FUNCTION_BLOCK PositionTrigger EXTENDS Objective

VAR
    internalPosition    	 : LREAL;
    internalTriggerDirection 	 : Tc2_MC2.MC_Direction;
    internalMoverPassedPosition : BOOL;
    internalCurrentMover     	 : POINTER TO Mover;
	internalLastMoverPassedPosition		: BOOL;
	internalTrack				: REFERENCE TO TRACK;
    moverLastPos              	: ARRAY[1..GVL.NUM_MOVERS] OF LREAL; // Positions of tracked movers from last cycle
	moverInitialized			: ARRAY [1..GVL.NUM_MOVERS] OF BOOL; // first scan-like flag to prevent erronious triggers on first scan
	
	lastCallMuteCurrent: LREAL;
	internalInterarrivalTimer			: TON;
	internalStatisticsReset				: BOOL;
END_VAR
VAR_OUTPUT
	Statistics							: PositionTriggerStats_typ;
END_VAR

{attribute 'monitoring' := 'call'}
PROPERTY CurrentMover : REFERENCE TO Mover
GET


CurrentMover						REF= internalCurrentMover^;
CurrentMover.SourceInstancePath		:= THIS^.InstancePath;

// If the Trigger has no CurrentMover, then return an imposter ErrorMover,
// whose method calls all trigger an error message
IF __ISVALIDREF(CurrentMover) = FALSE THEN
    ErrorMover.SourceInstancePath := THIS^.InstancePath;
    CurrentMover                  REF= ErrorMover;
END_IF
END_GET
END_PROPERTY

METHOD Cyclic : BOOL
VAR_INPUT
END_VAR
VAR
	
    i                       	: UDINT;	
	currentIsRegistered			: BOOL;
	moverTrackId				: INT;
	positionDifference			: LREAL;
	modTrackPosition			: LREAL;
	rolloverOccured				: BOOL;
	
END_VAR
VAR_INST

	velocityCount				: UDINT;
	velocitySum					: LREAL;
	internalRingBufferIDX		: UDINT;
	alphaEMA					: LREAL;

END_VAR
currentIsRegistered		:= FALSE;

FOR i := 1 TO GVL.NUM_MOVERS DO
    IF internalTrackedMovers[i] <> 0 AND_THEN internalTrackedMovers[i]^.IsTrackReady AND internalTrackedMovers[i]^.CurrentTrack <> 0 THEN
		moverTrackId := internalTrackedMovers[i]^.CurrentTrack^.Id;
		IF (moverTrackId = internalTrack.Id) THEN
			
			// last position is invalid on first scan, set it to the current position to avoid a false trigger on the first scan
			IF NOT moverInitialized[i] THEN
				moverInitialized[i] := TRUE;
				moverLastPos[i] := modTrackPosition;
			END_IF
		
			// Determine if a position rollover occured in the last cycle
			modTrackPosition := MODABS( internalTrackedMovers[i]^.TrackInfo.TrackPosition, internalTrackedMovers[i]^.CurrentTrack^.Length);
			positionDifference := moverLastPos[i] - modTrackPosition;			
			rolloverOccured := ABS( positionDifference ) > ( internalTrackedMovers[i]^.CurrentTrack^.Length / 2 );
			
			// and if so, modify the stored last position values to be nonmodulo to compensate
			IF rolloverOccured AND positionDifference > 0 THEN
				moverLastPos[i]		:= moverLastPos[i] - internalTrackedMovers[i]^.CurrentTrack^.Length;
			ELSIF rolloverOccured AND positionDifference < 0 THEN
				moverLastPos[i]		:= moverLastPos[i] + internalTrackedMovers[i]^.CurrentTrack^.Length;
			END_IF
		
			// Look for movers passing over the threshold this cycle and assign it to the
			// InternalCurrentMover output, which should latch until it is cleared
			IF TriggerDirection = MC_Positive_Direction AND moverLastPos[i] < internalPosition AND
				modTrackPosition >= internalPosition THEN
				
				// Position trigger event detected in the positive direction
				internalMoverPassedPosition		:= TRUE;
				internalCurrentMover			:= internalTrackedMovers[i];
				
			ELSIF TriggerDirection = MC_Negative_Direction AND moverLastPos[i] > internalPosition AND
				modTrackPosition <= internalPosition THEN
				
				// Position trigger event detecte in the negative direction
				internalMoverPassedPosition		:= TRUE;
				internalCurrentMover			:= internalTrackedMovers[i];
				
			END_IF
			
			
			
			// Ensure that the CurrentMover is still registered with the PositionTrigger
			IF internalCurrentMover <> 0 AND internalTrackedMovers[i] = internalCurrentMover THEN
				currentIsRegistered		:= TRUE;
			END_IF
	
			moverLastPos[i] 		:= modTrackPosition;
		END_IF
	END_IF

END_FOR


// If the CurrentMover isn't found in the registration list, then it has been removed, and should no longer be Current
IF currentIsRegistered = FALSE THEN
	internalMoverPassedPosition		:= FALSE;
	internalCurrentMover			:= 0;
END_IF

// Calculate stats
IF THIS^.MoverPassedPosition AND internalLastMoverPassedPosition = FALSE THEN
	// skip statistics on reset flag
	IF (internalStatisticsReset) THEN
		// reset flag
		internalStatisticsReset := FALSE;
		Statistics.ProcessedMoverCount									:= Statistics.ProcessedMoverCount + 1;
		// set weight of first mover to 1
		alphaEMA := 1.0;
	ELSE
		Statistics.ProcessedMoverCount									:= Statistics.ProcessedMoverCount + 1;
		Statistics.InterarrivalTimeHistory[internalRingBufferIDX]		:= internalInterarrivalTimer.ET;
		Statistics.MoverVelocityHistory[internalRingBufferIDX]			:= THIS^.CurrentMover.AxisReference.NcToPlc.ActVelo;
		internalRingBufferIDX											:= internalRingBufferIDX + 1;
		Statistics.LatestMoverVelocity									:= THIS^.CurrentMover.AxisReference.NcToPlc.ActVelo;
		Statistics.AverageInterarrivalTime	:= LREAL_TO_TIME(( alphaEMA * TIME_TO_LREAL(internalInterarrivalTimer.ET )) + (( 1 - alphaEMA) * TIME_TO_LREAL( Statistics.AverageInterarrivalTime )));
		internalInterarrivalTimer( IN := FALSE );
		// reset alphaema to global value for subsequent movers
		alphaEMA := GVL.ALPHA_EMA;
	END_IF;
END_IF
internalLastMoverPassedPosition		:= THIS^.MoverPassedPosition;
internalInterarrivalTimer( IN := NOT internalStatisticsReset, PT := T#40D, ET => Statistics.InterarrivalTime );

IF internalRingBufferIDX = ( SIZEOF( Statistics.InterarrivalTimeHistory ) / SIZEOF( Statistics.InterarrivalTimeHistory[0] )) THEN
	internalRingBufferIDX		:= 0;
END_IF

IF Statistics.AverageInterarrivalTime <> T#0S THEN
	Statistics.AverageMoversPerMinute		:= 60000 / TIME_TO_LREAL( Statistics.AverageInterarrivalTime );
END_IF

velocitySum		:= 0;
velocityCount	:= 0;

FOR i := 0 TO SIZEOF( Statistics.MoverVelocityHistory ) / SIZEOF( Statistics.MoverVelocityHistory[0] ) DO
	IF Statistics.MoverVelocityHistory[i] <> 0 THEN
		velocityCount		:= velocityCount + 1;
		velocitySum			:= velocitySum + Statistics.MoverVelocityHistory[i];
	END_IF
END_FOR
IF velocityCount <> 0 THEN // protect div0
	Statistics.AverageMoverVelocity		:= velocitySum / velocityCount;
END_IF
END_METHOD

{attribute 'monitoring' := 'call'}
PROPERTY MoverPassedPosition : BOOL
GET
MoverPassedPosition := internalMoverPassedPosition;
END_GET
END_PROPERTY

METHOD MuteCurrent : BOOL
VAR
	newCallTime			: LREAL;
END_VAR
VAR_INST
	MsgCreate			: FB_TcMessage;	
END_VAR
// message for debugging as this function is typically called when acting on a position trigger
newCallTime		:= ULINT_TO_LREAL(F_GetSystemTime())/1E7;
IF ( newCallTime - lastCallMuteCurrent ) > 1 THEN
	MsgCreate.CreateEx( TC_EVENTS.XtsBaseEventClass.PositionTriggerMuteCurrent,0 );
	MsgCreate.ipArguments.Clear().AddString(THIS^.InstancePath).AddUDint(internalCurrentMover^.IdentInGroup);
	MsgCreate.Send(0);
END_IF
lastCallMuteCurrent := newCallTime;

internalMoverPassedPosition		:= FALSE;
internalCurrentMover			:= 0;
END_METHOD

{attribute 'monitoring' := 'call'}
PROPERTY Position : LREAL
GET
Position := internalPosition;
END_GET
SET
// todo maybe do a limits check here?
internalPosition := Position;
END_SET
END_PROPERTY

METHOD ResetStatistics : BOOL
VAR_INPUT
END_VAR


Statistics.AverageInterarrivalTime		:= T#0S;
Statistics.AverageMoversPerMinute		:= 0;
Statistics.AverageMoverVelocity			:= 0;
Statistics.InterarrivalTime				:= T#0S;

memset(ADR(Statistics.InterarrivalTimeHistory),0,SIZEOF(Statistics.InterarrivalTimeHistory));
memset(ADR(Statistics.MoverVelocityHistory),0,SIZEOF(Statistics.MoverVelocityHistory));

Statistics.LatestMoverVelocity			:= 0;
Statistics.ProcessedMoverCount			:= 0;

internalStatisticsReset					:= TRUE;
END_METHOD

METHOD SetTrack : BOOL
VAR_INPUT
	Track : REFERENCE TO TRACK;
END_VAR
internalTrack REF= Track;
END_METHOD

PROPERTY TrackId : DINT
GET
TrackId := internalTrack.Id;
END_GET
END_PROPERTY

{attribute 'monitoring' := 'call'}
PROPERTY TriggerDirection : Tc2_MC2.MC_Direction
GET
TriggerDirection := internalTriggerDirection;
END_GET
SET
internalTriggerDirection := TriggerDirection;
END_SET
END_PROPERTY

END_FUNCTION_BLOCK

(* stored: Version 1.1.0.1, ProductVersion 3.1.4026.8
   POU PositionTrigger: Id {e261b23c-fca2-43e5-b385-fb66bc9fcaf5}, SpecialFunc None
   Folder Methods: Id {9cc02e33-a729-42f1-92ba-3e4f0abe5943}
   Folder Properties: Id {44d24ab5-188a-4889-a21d-6766b6bafebd}
   Property CurrentMover: Id {c163c3b6-4ffd-4a8a-9cd5-4f7ea2c9ac63}
   Get Get: Id {1ef15534-d318-4776-b5e9-9e8c1d9782f0}
   Method Cyclic: Id {4af842ce-a8b8-45a8-81bc-ac521b0a027a}
   Property MoverPassedPosition: Id {a772009e-789b-4c33-900b-53697bdea9b4}
   Get Get: Id {609e4250-8b2f-45f6-8a69-75a39f309494}
   Method MuteCurrent: Id {39742f47-b11e-053a-08ba-d3a07a9ed4a0}
   Property Position: Id {25b3d396-dcf1-4a9a-afb5-cc0f915e5828}
   Get Get: Id {36b155cf-1e07-48aa-8c28-02916d4da719}
   Set Set: Id {7efc021c-c389-4be4-95cc-10506809ec26}
   Method ResetStatistics: Id {485f63f0-075c-0e7c-1416-0b610b27218f}
   Method SetTrack: Id {1692464a-54c2-0d6f-250a-480aa9560f30}
   Property TrackId: Id {dbfe845b-02ea-002a-11b5-4efaf37a2e66}
   Get Get: Id {36306272-b6fe-0043-1e2d-da060775dff6}
   Property TriggerDirection: Id {13bb661c-6cea-4df5-a26e-19ba5cdbbe66}
   Get Get: Id {8bbc3265-3408-4a78-8182-d12cc43c4309}
   Set Set: Id {3c003fcd-3a77-441b-81df-74705c2d0fc5} *)
